// TIA Portal V21 export
VAR_GLOBAL   // PLC tag table "K_TipoAnalogica"
END_VAR
VAR_GLOBAL CONSTANT   // user constants
   K_TipoAnalogicaEw : Int := 0;
   K_TipoAnalogicaProfinetHendressHauser : Int := 1;
   K_TipoAnalogicaSondeDigitali : Int := 2;
   K_TipoAnalogicaViaReteS7 : Int := 3;
END_VAR
